{attribute 'GeneratedUsingTerminal: EP3744-0041-0016'}
{attribute addProperty BoxType "EP3744-0041-0016"}
{attribute addProperty Id "InputAT %I*ARRAY[0..5] OF BOOL6"}
{attribute addProperty CRC "390650255"}
{attribute addProperty Size "6"}
TYPE DIG_Inputs_697E0EF2 :
STRUCT
	{attribute addProperty Name "Input"}
	Input AT %I* : ARRAY[0..5] OF BOOL;
END_STRUCT
END_TYPE

(* stored: Version 1.2.0.0, ProductVersion 3.1.4024.9
   DUT DIG_Inputs_697E0EF2: Id {92ce7630-1824-4e73-8471-b45d1c90e78e} *)
